RoboDK station: Final_simulation.rdk

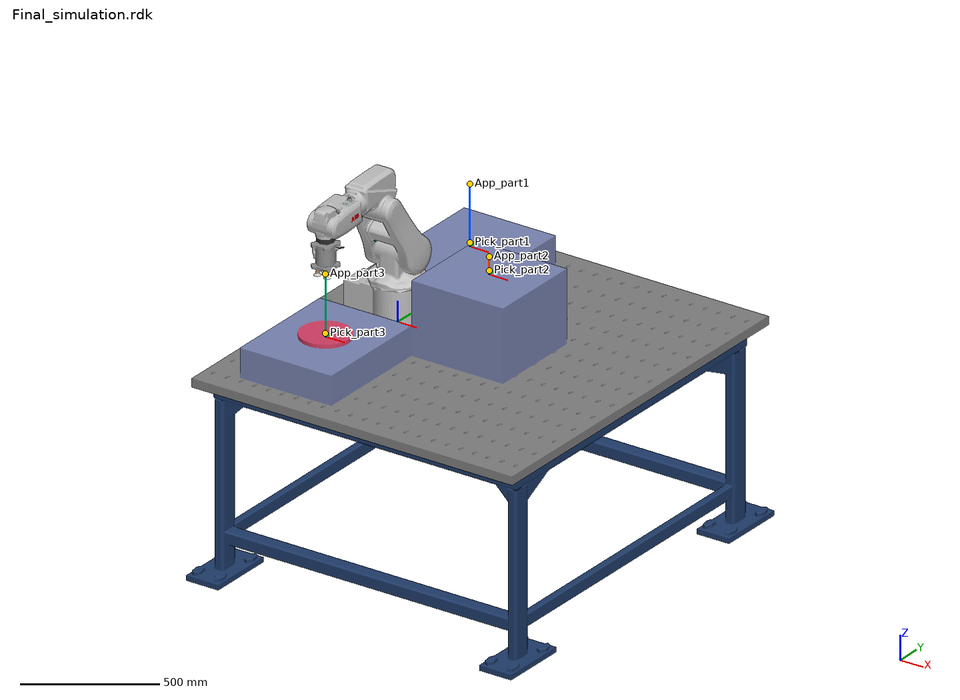
[picture v0: the station drawn from its stored meshes, robots at their saved joint values, targets as dots, program paths as lines]
Station Final (saved by RoboDK 5.6.2). Poses are relative to the parent item; angles as X-Y-Z fixed-axis rotations.
  - object Table 1400x800x800mm at (0, 0, 0) mm, size 1420 x 1640 x 800 mm, geometry from Table-1400x800x800mm.sld
  - frame ABB IRB 120-3/0.6 Base at (0, 0, 0) mm
    - robot ABB IRB 120-3/0.6: 6 axes, payload 3 kg, reach 580 mm, repeatability 0.01 mm, weight 25 kg
        modified DH rows (alpha deg, a mm, theta deg, d mm): 0, 0, 0, 290; -90, 0, -90, 0; 0, 270, 0, 0; -90, 70, 0, 302; 90, 0, 0, 0; -90, 0, 180, 72
        joint limits [-165, -110, -90, -160, -120, -400] to [165, 110, 70, 160, 120, 400]; home [0, 0, 0, 0, 0, 0]; saved at [-90, 32.183, -28.131, 0, 85.948, 0]
      - tool SMC ZXP7A01-ZP25C-X1 Vacuum Gripper, TCP at (0, 0, 125) mm, size 88 x 106.8 x 127.9 mm
  - object object1 at (400, 0, 0) mm, size 400 x 400 x 300 mm, geometry from object1.STEP
  - object object2 at (0, 450, 60) mm, size 400 x 500 x 120 mm, geometry from object2.STEP
  - object object3 at (0, -450, 60) mm, size 400 x 500 x 120 mm, geometry from object2.STEP
  - frame part_1 at (0, 450, 120) mm
    - target App_part1 (Cartesian target) at (0, 0, 250) mm, rotated rx 180 ry 0 rz -90 deg; joints [90, 32.183, -28.131, 0, 85.948, 0] of ABB IRB 120-3/0.6
    - target Pick_part1 (Cartesian target) at (0, 0, 14) mm, rotated rx 180 ry 0 rz -90 deg; joints [90, 42.67, 0.92, 0, 46.411, 0] of ABB IRB 120-3/0.6
  - frame part_2 at (400, 0, 300) mm
    - target App_part2 (Cartesian target) at (0, 0, 70) mm, rotated rx 180 ry 0 rz -180 deg; joints [0, 19.658, -10.814, 0, 81.156, 0] of ABB IRB 120-3/0.6
    - target Pick_part2 (Cartesian target) at (0, 0, 15) mm, rotated rx 180 ry 0 rz -180 deg; joints [0, 19.842, -0.873, 0, 71.031, 0] of ABB IRB 120-3/0.6
  - frame part_3 at (0, -450, 120) mm
    - target App_part3 (Cartesian target) at (0, 0, 250) mm, rotated rx 180 ry 0 rz 90 deg; joints [-90, 32.183, -28.131, 0, 85.948, 0] of ABB IRB 120-3/0.6
    - target Pick_part3 (Cartesian target) at (0, 0, 15) mm, rotated rx 180 ry 0 rz 90 deg; joints [-90, 42.56, 0.891, 0, 46.55, 0] of ABB IRB 120-3/0.6
  - program ReplaceObjects (1 instructions, listed below)
  - program Pick_1 (6 instructions, listed below)
  - program Pick_2 (9 instructions, listed below)
  - program Pick_3 (6 instructions, listed below)
  - program MainProgram (4 instructions, listed below)
  - object Cylinder 50x150mm at (0, -450, 121) mm, rotated rx 0 ry 0 rz 180 deg, size 200 x 200 x 15 mm, geometry from Cylinder-50x150mm.sld
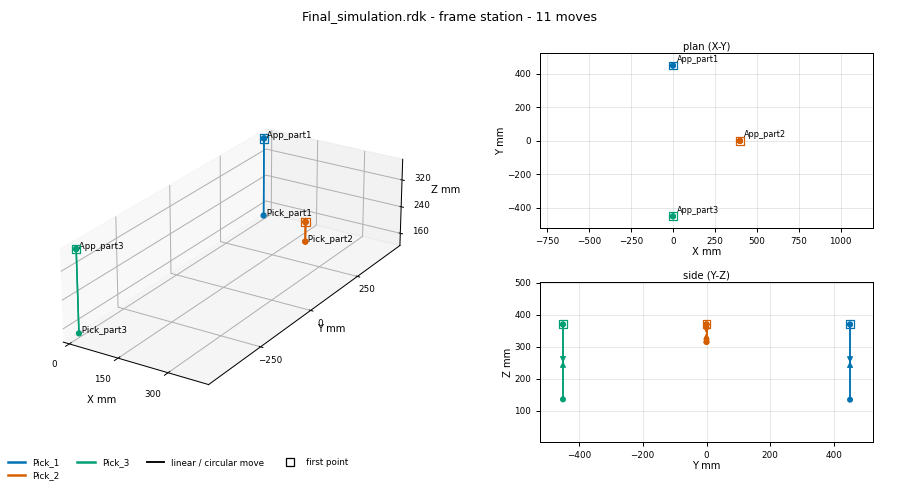
[picture p0: tool path of Final_simulation.rdk in frame station, 11 of 11 moves have a stored position in this frame; points joined in program order, loops and branches not executed]

--- program ReplaceObjects (robot ABB IRB 120-3/0.6) ---
  Replace objects

--- program Pick_1 (robot ABB IRB 120-3/0.6) ---
  Set Ref.: part_1
  Set Tool: SMC ZXP7A01-ZP25C-X1 Vacuum Gripper
  MoveJ (App_part1)
  MoveL (Pick_part1)
  Attach to SMC ZXP7A01-ZP25C-X1 Vacuum Gripper
  MoveL (App_part1)

--- program Pick_2 (robot ABB IRB 120-3/0.6) ---
  Set Ref.: part_2
  Set Tool: SMC ZXP7A01-ZP25C-X1 Vacuum Gripper
  MoveJ (App_part2)
  MoveL (Pick_part2)
  Detach from SMC ZXP7A01-ZP25C-X1 Vacuum Gripper
  MoveL (App_part2)
  MoveL (Pick_part2)
  Attach to SMC ZXP7A01-ZP25C-X1 Vacuum Gripper
  MoveL (App_part2)

--- program Pick_3 (robot ABB IRB 120-3/0.6) ---
  Set Ref.: part_3
  Set Tool: SMC ZXP7A01-ZP25C-X1 Vacuum Gripper
  MoveJ (App_part3)
  MoveL (Pick_part3)
  Detach from SMC ZXP7A01-ZP25C-X1 Vacuum Gripper
  MoveL (App_part3)

--- program MainProgram (robot ABB IRB 120-3/0.6) ---
  Call ReplaceObjects
  Call Pick_1
  Call Pick_2
  Call Pick_3
